Staubli VAL3: onF2Event.pgx

program onF2Event()
  local string l_sItem
begin
 // look if the bButton is enable
  call loadPage("instrSequential/AXIS7/page_axis",l_sItem)
end
